TEXTLIST TL_FbState
  0 = 'UNDEFINED'
  1 = 'RUN'
  2 = 'STOP'
  3 = 'SAFE'
  4 = 'ERROR'
  5 = 'RESET'
  6 = 'START'
  7 = 'ERROR DELAY'
  8 = 'DELAY OUT'
  9 = 'FUNC TEST'
  11 = '1 BUTTON'
  12 = '2 BUTTON'
  13 = 'REALISE'
  14 = 'MON OFF'
  15 = 'MON ON'
   = ''
END_TEXTLIST

(* stored: Version 1.1.0.1, ProductVersion 3.1.4022.12
   TextList TL_FbState: Id {f5f993f9-f906-4098-8036-fd7b0a321d32} *)
